INTERFACE ITestOperation EXTENDS __SYSTEM.IQueryInterface

METHOD AssertEqual
VAR_INPUT
	Var1					: ANY;
	Var2					: ANY;
	FloatingPointTollerance : LREAL := 0.000001;
END_VAR
END_METHOD

METHOD ExecuteTest : BOOL
VAR_INPUT
END_VAR
END_METHOD

PROPERTY State : E_TestStatus
GET
END_GET
SET
END_SET
END_PROPERTY

PROPERTY TestId : T_MaxString
GET
END_GET
SET
END_SET
END_PROPERTY

END_INTERFACE

(* stored: Version 1.1.0.1
   Itf ITestOperation: Id {08860d6e-c469-4ecd-9c53-2cb76abc1038}
   Method AssertEqual: Id {9c1c2102-a6cd-43d4-b955-8a4e23076c37}
   Method ExecuteTest: Id {b962dfa9-06a4-472e-bbe7-928854d9dd2a}
   Property State: Id {15265f80-3995-432c-9bc2-2c1127cdc374}
   Get Get: Id {addd4951-db3c-4ab4-85c4-bed3a300a2e3}
   Set Set: Id {09f71b2a-b665-430b-932e-7ad90451fb6e}
   Property TestId: Id {7a2b531b-1e78-4625-bf6c-a530812e3b3e}
   Get Get: Id {36d24df8-a9ee-41ce-b400-8b72587288f6}
   Set Set: Id {daf96dcf-8df8-4e4e-9750-a5d6e2a7dff9} *)
